PROGRAM main
  VAR
    timer_1s : TON; (* 1秒週期計時器 *)
    pulse_1s : BOOL; (* 每秒一個掃描周期的脈衝 *)
    counter_1 : CTU; (* 加計記數器 *)
    counter_value AT %QW0 : INT; (* 計數值，要給Modbus讀 *)
    counter_full : BOOL; (* 計數到達預設值 *)
    counter_limit AT %QW1 : INT; (* 計數器上限 *)
    effective_limit AT %QW2 : INT;
  END_VAR

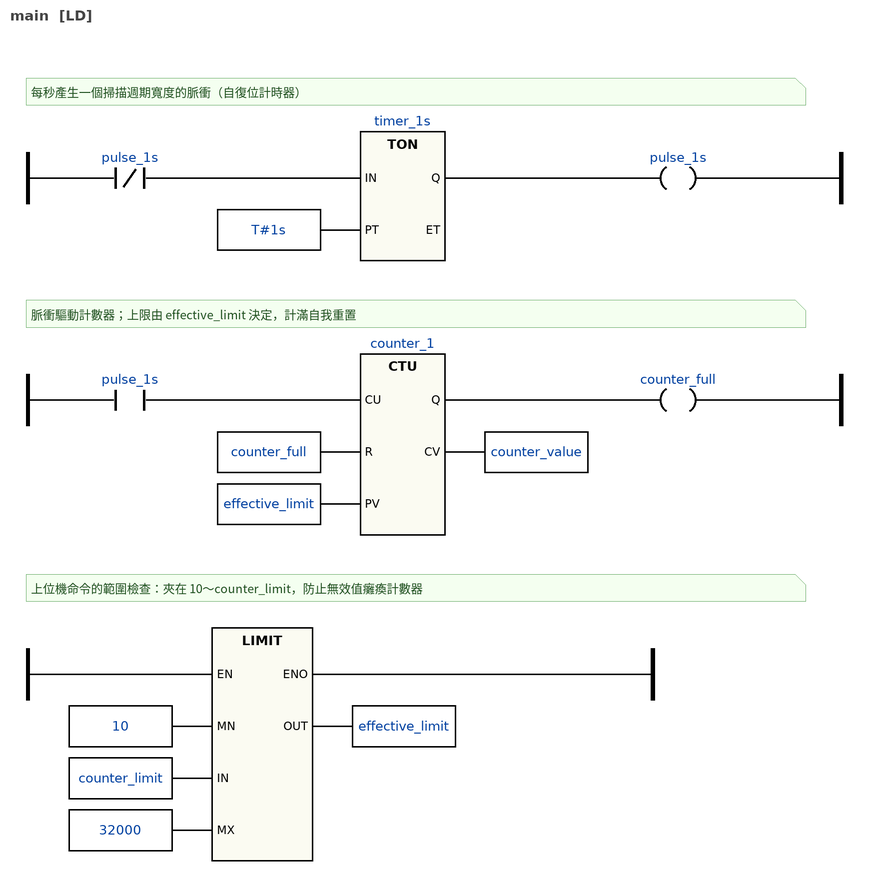
(* LD diagram, written out as Structured Text *)
(* 每秒產生一個掃描週期寬度的脈衝（自復位計時器） *)
timer_1s(IN := NOT pulse_1s, PT := T#1s);
pulse_1s := timer_1s.Q;
(* 脈衝驅動計數器；上限由 effective_limit 決定，計滿自我重置 *)
counter_1(CU := pulse_1s, R := counter_full, PV := effective_limit);
counter_full := counter_1.Q;
counter_value := counter_1.CV;
(* 上位機命令的範圍檢查：夾在 10～counter_limit，防止無效值癱瘓計數器 *)
effective_limit := LIMIT(10, counter_limit, 32000);
END_PROGRAM
